Staubli VAL3: MX1_NETWORK.pjx

--- MX1_NETWORK.pjx ---
Parameters version=s7.9.4 stackSize=5000 millimeterUnit=true
Program file=argumentParse.pgx
Program file=commandCheck.pgx
Program file=commandExecute.pgx
Program file=dataReset.pgx
Program file=ioLinks.pgx
Program file=serverCmd.pgx
Program file=socketRead.pgx
Program file=socketWrite.pgx
Program file=start.pgx
Program file=stop.pgx
Data file=MX1_NETWORK.dtx
Library alias=MX1_COMMANDS path=Disk://MX1_COMMANDS autoload=true password=
Library alias=io path=Disk://io autoload=true password=

--- MX1_NETWORK.dtx ---
mdesc mNomSpeed
sio sSocket1 = {link=Socket\sock1}

--- start.pgx ---
program start()
begin
  call ioLinks()
  taskCreate "network",100,serverCmd()
end

--- argumentParse.pgx ---
program argumentParse(num& nBuffer[] (dimensions=1), num nBytes (dimensions=1), num& nArgs[] (dimensions=1), num& nNbArgs (dimensions=1), string& sBuffer (dimensions=1), string& sCommand (dimensions=1))
  local bool bFlag
  local num nIndex
  local num ni
begin
  //convert to string and parse socket data
  sBuffer=""
  //CONVERT TO STRING
  for ni=0 to (nBytes-1) step 1
    sBuffer=sBuffer+chr(nBuffer[ni])
  endFor
  //GET COMMAND NAME
  sCommand=""
  nNbArgs=0
  nIndex=find(sBuffer," ")
  if nIndex==-1
    //command without arguments
    sCommand=sBuffer
  else
    //command with arguments
    sCommand=left(sBuffer,nIndex)
    //GET ARGUMENTS
    //skip space right side characters
    sBuffer=right(sBuffer,nBytes-len(sCommand)-1)
    while (asc(sBuffer,0)==32) and (len(sBuffer)>0)
      sBuffer=right(sBuffer,len(sBuffer)-1)
    endWhile
    //extract arguments
    bFlag=false
    do
      sBuffer=toNum(sBuffer,nArgs[nNbArgs],bFlag)
      nNbArgs=nNbArgs+1
    until (bFlag!=true) or (nNbArgs>8)
    nNbArgs=nNbArgs-1
  endIf
end

--- commandCheck.pgx ---
program commandCheck(num& nArgs[] (dimensions=1), num nNbArgs (dimensions=1), string& sBuffer (dimensions=1), string sCommand (dimensions=1), bool& bFlag (dimensions=1))
begin
  //check command name and arguments
  //everything passed by reference from serverCmd
  bFlag=false
  switch sCommand
    case "gripper"
      if nNbArgs!=1
        sBuffer="NACK: "+sCommand+" nNbArgs: "+chr(nNbArgs)
      else
        if (nArgs[0]<0) or (nArgs[0]>1)
          sBuffer="NACK: "+sCommand+" nArgs[0]: "+chr(nArgs[0])
        else
          bFlag=true
        endIf
      endIf
    break
    case "power"
      if nNbArgs!=1
        sBuffer="NACK: "+sCommand+" nNbArgs: "+toString("",nNbArgs)
      else
        if (nArgs[0]<0) or (nArgs[0]>1)
          sBuffer="NACK: "+sCommand+" nArgs[0]: "+toString("",nArgs[0])
        else
          bFlag=true
        endIf
      endIf
    break
    case "stopMove"
      if nNbArgs!=0
        sBuffer="NACK: "+sCommand+" nNbArgs: "+chr(nNbArgs)
      else
        bFlag=true
      endIf
    break
    case "restartMove"
      if nNbArgs!=0
        sBuffer="NACK: "+sCommand+" nNbArgs: "+chr(nNbArgs)
      else
        bFlag=true
      endIf
    break
    case "isSettled"
      if nNbArgs!=0
        sBuffer="NACK: "+sCommand+" nNbArgs: "+chr(nNbArgs)
      else
        bFlag=true
      endIf
    break
    case "setFrame"
      if nNbArgs!=1
        sBuffer="NACK: "+sCommand+" nNbArgs: "+chr(nNbArgs)
      else
        if (nArgs[0]<0) or (nArgs[0]>3)
          sBuffer="NACK: "+sCommand+" nArgs[0]: "+chr(nArgs[0])
        else
          bFlag=true
        endIf
      endIf
    break
    case "setTool"
      if nNbArgs!=1
        sBuffer="NACK: "+sCommand+" nNbArgs: "+chr(nNbArgs)
      else
        if (nArgs[0]<0) or (nArgs[0]>3)
          sBuffer="NACK: "+sCommand+" nArgs[0]: "+chr(nArgs[0])
        else
          bFlag=true
        endIf
      endIf
    break
    case "moveX"
      if nNbArgs!=1
        sBuffer="NACK: "+sCommand+" nNbArgs: "+chr(nNbArgs)
      else
        if abs(nArgs[0])>50
          sBuffer="NACK: "+sCommand+" nArgs[0]: "+chr(nArgs[0])
        else
          bFlag=true
        endIf
      endIf
    break
    case "moveY"
      if nNbArgs!=1
        sBuffer="NACK: "+sCommand+" nNbArgs: "+chr(nNbArgs)
      else
        if abs(nArgs[0])>50
          sBuffer="NACK: "+sCommand+" nArgs[0]: "+chr(nArgs[0])
        else
          bFlag=true
        endIf
      endIf
    break
    case "moveZ"
      if nNbArgs!=1
        sBuffer="NACK: "+sCommand+" nNbArgs: "+chr(nNbArgs)
      else
        if abs(nArgs[0])>50
          sBuffer="NACK: "+sCommand+" nArgs[0]: "+chr(nArgs[0])
        else
          bFlag=true
        endIf
      endIf
    break
    case "getX"
      if nNbArgs!=0
        sBuffer="NACK: "+sCommand+" nNbArgs: "+chr(nNbArgs)
      else
        bFlag=true
      endIf
    break
    case "getY"
      if nNbArgs!=0
        sBuffer="NACK: "+sCommand+" nNbArgs: "+chr(nNbArgs)
      else
        bFlag=true
      endIf
    break
    case "getZ"
      if nNbArgs!=0
        sBuffer="NACK: "+sCommand+" nNbArgs: "+chr(nNbArgs)
      else
        bFlag=true
      endIf
    break
    default
      logMsg("commandCheck fail: "+sCommand)
    break
  endSwitch
  //
end

--- commandExecute.pgx ---
program commandExecute(num& nArgs[] (dimensions=1), num nNbArgs (dimensions=1), string& sBuffer (dimensions=1), string sCommand (dimensions=1))
  local num nGetArg1
  local num nGetArg2
begin
  //execute command stored in global variables
  //bFlag check must be done previously in start()
  switch sCommand
    case "gripper"
      call MX1_COMMANDS:gripper(nArgs[0])
      sBuffer="ACK: "+sCommand+" "+toString("",nArgs[0])
    break
    case "power"
      call MX1_COMMANDS:power(nArgs[0])
      sBuffer="ACK: "+sCommand+" "+toString("",nArgs[0])
    break
    case "stopMove"
      call MX1_COMMANDS:stopMove()
      //stopMove()
      sBuffer="ACK: "+sCommand
    break
    case "restartMove"
      call MX1_COMMANDS:restartMove()
      //restartMove()
      sBuffer="ACK: "+sCommand
    break
    case "isSettled"
      call MX1_COMMANDS:isSettled(nGetArg1)
      //bGetArg1 = isSettled()
      sBuffer="ACK: "+sCommand+" "+toString("",nGetArg1)
    break
    case "setFrame"
      call MX1_COMMANDS:setFrame(nArgs[0])
      sBuffer="ACK: "+sCommand+" "+toString("",nArgs[0])
    break
    case "setTool"
      call MX1_COMMANDS:setTool(nArgs[0])
      sBuffer="ACK: "+sCommand+" "+toString("",nArgs[0])
    break
    case "moveX"
      call MX1_COMMANDS:moveX(nArgs[0])
      sBuffer="ACK: "+sCommand+" "+toString("",nArgs[0])
    break
    case "moveY"
      call MX1_COMMANDS:moveY(nArgs[0])
      sBuffer="ACK: "+sCommand+" "+toString("",nArgs[0])
    break
    case "moveZ"
      call MX1_COMMANDS:moveZ(nArgs[0])
      sBuffer="ACK: "+sCommand+" "+toString("",nArgs[0])
    break
    case "getX"
      call MX1_COMMANDS:getX(nGetArg1)
      sBuffer="ACK: "+sCommand+" "+toString(".3",nGetArg1)
    break
    case "getY"
      call MX1_COMMANDS:getY(nGetArg1)
      sBuffer="ACK: "+sCommand+" "+toString(".3",nGetArg1)
    break
    case "getZ"
      call MX1_COMMANDS:getZ(nGetArg1)
      sBuffer="ACK: "+sCommand+" "+toString(".3",nGetArg1)
    break
    default
      logMsg("commandExecute fail: "+sCommand)
    break
  endSwitch
end

--- dataReset.pgx ---
program dataReset()
  local num ni
begin
  clearBuffer(sSocket1)
end

--- ioLinks.pgx ---
program ioLinks()
begin
  //link sock1 - J204 to sSocket sio
  sioLink(sSocket1,io:sock1)
end

--- serverCmd.pgx ---
program serverCmd()
  local bool bFlag
  local num nArgs[8]
  local num nBuffer[30]
  local num nBytes
  local num nIndex
  local num nNbArgs
  local num ni
  local string sBuffer
  local string sCommand
begin
  //server task - read and write on socket
  //SETUP - CLEAR BUFFER
  clearBuffer(sSocket1)
  ////////FOREVER LOOP - TASK////////
  while (true)
    //nBytes = number of bytes read to nBuffer
    //nBytes must be less than 30 and not empty
    nBytes=sioGet(sSocket1,nBuffer)
    if (nBytes>0) and (nBytes<30)
      //INPUT PARSING
      call argumentParse(nBuffer,nBytes,nArgs,nNbArgs,sBuffer,sCommand)
      //CHECK COMMAND
      call commandCheck(nArgs,nNbArgs,sBuffer,sCommand,bFlag)
      if bFlag==true
        //EXECUTE COMMAND
        call commandExecute(nArgs,nNbArgs,sBuffer,sCommand)
      else
        logMsg("serverCmd: bFlag == false")
      endIf
      //OUTPUT WRITE
      call socketWrite(sBuffer,nBuffer)
      nBytes=sioSet(sSocket1,nBuffer)
      if (nBytes<0)
        logMsg("serverCmd: sioSet error > "+toString("",nBytes))
      endIf
    else
      logMsg("serverCmd: sioget error > "+chr(nBytes))
    endIf
  endWhile
end

--- socketRead.pgx ---
program socketRead()
begin
end

--- socketWrite.pgx ---
program socketWrite(string& sBuffer (dimensions=1), num& nBuffer[] (dimensions=1))
  local num ni
begin
  if len(sBuffer)>29
    sBuffer=left(sBuffer,29)
  endIf
  for ni=0 to 29 step 1
    nBuffer[ni]=0
  endFor
  for ni=0 to (len(sBuffer)-1) step 1
    nBuffer[ni]=asc(sBuffer,ni)
  endFor
  nBuffer[ni]=13
end
